FUNCTION_BLOCK FB_CylinderTempRecord EXTENDS FB_CylinderTemp
VAR_INPUT
	bRecordStart				:	BOOL;							// Signal to start recording temperature
	nTimeInterval				:	TIME;							// Time interval between samples of temperature
END_VAR
VAR_OUTPUT
	bRecordFullDone				:	BOOL;							// TRUE if the temperature recording is done
	aRecords					:	ARRAY [1..100] OF	LREAL;		//	Array with temperature records
END_VAR
VAR
	nIndex						:	UDINT;							// Index to handle temperature array
	fbTimerInterval				:	TON;							// Timer to control the recording interval
END_VAR

// ===================================================================
;
// ===================================================================

METHOD Record
VAR_INPUT
END_VAR

	bRecordFullDone := (nIndex := 100);

	IF bRecordStart AND NOT bRecordFullDone AND NOT fbTimerInterval.Q THEN
		fbTimerInterval(	IN		:=		TRUE,
							PT		:=		fbTimerInterval);
	END_IF
	
	IF fbTimerInterval.Q THEN
		fbTimerInterval(	IN		:=		FALSE);
		
		nIndex					:=		nIndex + 1;
		aRecords[nIndex]		:=		fTempCurrent;
	END_IF
END_METHOD

METHOD Reset
VAR_INPUT
END_VAR
	SUPER^.Reset();

	FOR nIndex	:= 1 TO 100 BY 1 DO
		aRecords[nIndex]	:=	0;
	END_FOR

	nIndex		:= 		0;
END_METHOD

END_FUNCTION_BLOCK

(* stored: Version 1.1.0.1, ProductVersion 3.1.4024.15
   POU FB_CylinderTempRecord: Id {663cafa0-e5e6-4d81-a8fe-461c8f79e9a1}, SpecialFunc None
   Method Record: Id {b629170c-9f79-4b11-9032-d566512463bc}
   Method Reset: Id {be66d682-a1e9-4c53-9139-cb671f3b3da7} *)
